// TIA Portal project "babu_switchPbLatestRecognize" (V15)

(* hardware
DEVICE "S7-1200 station_1"  S7-1200 Station
   slot 0: "Rack_0"  S7-1200 Rack  Rack  V1.0
   slot 1: "PLC_1"  CPU 1212C DC/DC/DC  6ES7 212-1AE40-0XB0  V4.2
*)

// ===== PLC "PLC_1"  CPU 1212C DC/DC/DC =====

VAR_GLOBAL   // PLC tag table "Tag table_1"
   "S1" AT %M0.0 : Bool;
   "F1" AT %M0.1 : Bool;
   "P1" AT %M0.2 : Bool;
   "M1" AT %M0.3 : Bool;
END_VAR

ORGANIZATION_BLOCK "Main"   // OB1, LAD, ProgramCycle
TITLE = "Main Program Sweep (Cycle)"
{ S7_Optimized_Access := 'TRUE' }
VERSION : 0.1
   VAR_INPUT
      Initial_Call : Bool;   // Initial call of this OB
      Remanence : Bool;   // =True, if remanent data are available
   END_VAR
BEGIN

REGION Network 1
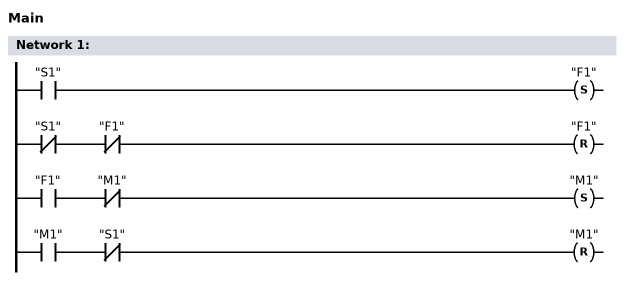
   RUNG wire#powerrail
      Contact( "S1" )
      S_Coil( "F1" )
   END_RUNG
   RUNG wire#powerrail
      I_Contact( "S1" )
      I_Contact( "F1" )
      R_Coil( "F1" )
   END_RUNG
   RUNG wire#powerrail
      Contact( "F1" )
      I_Contact( "M1" )
      S_Coil( "M1" )
   END_RUNG
   RUNG wire#powerrail
      Contact( "M1" )
      I_Contact( "S1" )
      R_Coil( "M1" )
   END_RUNG
   // the same network as SCL:
   IF "S1" THEN "F1" := TRUE; END_IF;
   IF NOT "S1" AND NOT "F1" THEN "F1" := FALSE; END_IF;
   IF "F1" AND NOT "M1" THEN "M1" := TRUE; END_IF;
   IF "M1" AND NOT "S1" THEN "M1" := FALSE; END_IF;
END_REGION
END_ORGANIZATION_BLOCK